FUNCTION_BLOCK WaterMonitorSensor_HCECC (* Model a conveyor *)
  (* Standard: 61499-2 *)
  (* Version 0.2, 2003-12-04, JHC, Rockwell Automation, Renamed for better indexing. *)
  (* Compiler header: package fb.rt.benchmarks.watermonitor; *)
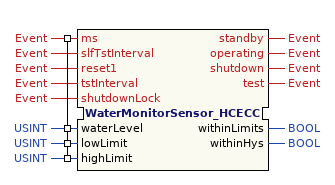
  EVENT_INPUT
    ms WITH waterLevel, lowLimit, highLimit; (* millisecond *)
    slfTstInterval;
    reset1;
    tstInterval;
    shutdownLock;
  END_EVENT
  EVENT_OUTPUT
    standby;
    operating;
    shutdown;
    test;
  END_EVENT
  VAR_INPUT
    waterLevel : USINT := 150;
    lowLimit : USINT := 100;
    highLimit : USINT := 200;
  END_VAR
  VAR_OUTPUT
    withinLimits : BOOL := true;
    withinHys : BOOL := true;
  END_VAR
  ALGORITHM inHys IN ST: (* Normally executed algorithm *)
withinHys := TRUE;
withinLimits := TRUE;
  END_ALGORITHM
  ALGORITHM outHys IN ST:
withinHys := FALSE;
  END_ALGORITHM
  ALGORITHM inLimits IN ST: (* Initialization algorithm *)
withinLimits := TRUE;
  END_ALGORITHM
  ALGORITHM outLimits IN ST:
withinLimits := FALSE;
withinHys := FALSE;
  END_ALGORITHM
END_FUNCTION_BLOCK
(* other elements stored in the file *)
(* ECC Name=Sensor *)
(* ECState Name=START Comment=Initial State *)
(* ECState Name=INHYS Comment=in hysterisis *)
(* ECAction Algorithm=inHys *)
(* ECState Name=INLIMITS Comment=within limts *)
(* ECState Name=OUTLIMITS Comment=outside limits *)
(* ECState Name=OUTHYS Comment=outside hysterisis *)
(* ECTransition Source=START Destination=INHYS Condition=ms&(waterLevel>(lowLimit+5) and waterLevel<(highLimit-5)) *)
(* ECTransition Source=START Destination=OUTHYS Condition=ms&(waterLevel<=(lowLimit+5) or waterLevel>=(highLimit-5)) *)
(* ECTransition Source=START Destination=INLIMITS Condition=ms&(waterLevel>lowLimit and waterLevel<highLimit) *)
(* ECTransition Source=START Destination=OUTLIMITS Condition=ms&(waterLevel<=lowLimit or waterLevel>=highLimit) *)
(* ECTransition Source=INHYS Destination=OUTHYS Condition=ms&(waterLevel<=(lowLimit+5) or waterLevel>=(highLimit-5)) *)
(* ECTransition Source=OUTHYS Destination=INHYS Condition=ms&(waterLevel>(lowLimit+5) and waterLevel<(highLimit-5)) *)
(* ECTransition Source=OUTHYS Destination=INLIMITS Condition=ms&(waterLevel>lowLimit and waterLevel<highLimit) *)
(* ECTransition Source=INLIMITS Destination=OUTHYS Condition=ms&(waterLevel<=(lowLimit+5) or waterLevel>=(highLimit-5)) *)
(* ECTransition Source=INLIMITS Destination=OUTLIMITS Condition=ms&(waterLevel<=lowLimit or waterLevel>=highLimit) *)
(* ECTransition Source=OUTLIMITS Destination=INLIMITS Condition=ms&(waterLevel>lowLimit and waterLevel<highLimit) *)
(* ECC Name=Monitor *)
(* ECState Name=STANDBY Comment=Initial State *)
(* ECState Name=SHUTDOWN *)
(* ECAction Output=shutdown *)
(* ECState Name=OPERATING *)
(* ECAction Output=operating *)
(* ECState Name=TEST *)
(* ECAction Output=test *)
(* ECTransition Source=STANDBY Destination=TEST Condition=slfTstInterval *)
(* ECTransition Source=STANDBY Destination=OPERATING Condition=reset1&withinLimits *)
(* ECTransition Source=TEST Destination=TEST Condition=slfTstInterval *)
(* ECTransition Source=TEST Destination=STANDBY Condition=tstInterval *)
(* ECTransition Source=OPERATING Destination=TEST Condition=slfTstInterval *)
(* ECTransition Source=OPERATING Destination=SHUTDOWN Condition=not withinLimits *)
(* ECTransition Source=SHUTDOWN Destination=TEST Condition=slfTstInterval *)
(* ECTransition Source=SHUTDOWN Destination=OPERATING Condition=withinHys *)
(* ECTransition Source=SHUTDOWN Destination=STANDBY Condition=shutdownLock *)
